INTERFACE ITF_Electrovalve_HMI_Connector EXTENDS ITF_BaseComponent_HMI_Connector

METHOD PUBLIC GetElectrovalveType : E_ElectrovalveType
VAR_INPUT
END_VAR
END_METHOD

METHOD PUBLIC GetElectrovalveTypeToString : STRING
END_METHOD

METHOD IsActiveCoilA : BOOL
VAR_INPUT
END_VAR
END_METHOD

METHOD IsActiveCoilB : BOOL
VAR_INPUT
END_VAR
END_METHOD

END_INTERFACE

(* stored: Version 1.1.0.1
   Itf ITF_Electrovalve_HMI_Connector: Id {d4a986f2-1106-4bb3-b7ec-204a8112af04}
   Method GetElectrovalveType: Id {6e27c53d-ec2e-4987-af63-a8db74574041}
   Method GetElectrovalveTypeToString: Id {8a63f63e-e75e-4d5c-83ff-12a7545b7d20}
   Method IsActiveCoilA: Id {11b33871-a6df-4b90-baea-ec7b047b3044}
   Method IsActiveCoilB: Id {f4705d69-b065-4cba-b1f2-d89d38866ff5} *)
